// TIA Portal project "FB CONTADOR" (V11)

(* hardware
DEVICE "S7300/ET200 station_1"  SIMATIC 300-Station
   slot 0: "Perfil soporte_0"  Rail  6ES7 390-1***0-0AA0
   slot 1: "PS 307 2A_1"  PS 307 2A  6ES7 307-1BA00-0AA0
   slot 2: "PLC_1"  CPU 313C-2 DP  6ES7 313-6CF03-0AB0  V2.6
      slot 0: "Interfaz MPI_1"  MPI
      slot 1: "Interfaz DP_1"  DP
      slot 2: "DI16/DO16_1"  DI16/DO16
      slot 4: "Contaje_1"  Counter
   slot 4: "AI4/AO2 x 8bits_1"  AI4/AO2x8/8Bit  6ES7 334-0CE01-0AA0
   slot 5: "CP 343-1 Lean_1"  CP 343-1 LEAN  6GK7 343-1CX10-0XE0  V2.4
   slot 6: "CP 340 RS232C_1"  CP 340 RS232C  6ES7 340-1AH02-0AE0  V1.0
   slot 7: "CP 340 RS422/485_2"  CP 340 RS422/485  6ES7 340-1CH02-0AE0  V1.0
*)

// ===== PLC "PLC_1"  CPU 313C-2 DP =====

VAR_GLOBAL   // PLC tag table "Tabla de variables estándar"
   "MARCHA" AT %E0.0 : Bool;
   "PARO" AT %E0.1 : Bool;
   "OUT" AT %A0.0 : Bool;
   "Tag_1" AT %E0.2 : Bool;
   "Tag_2" AT %T0 : Timer;
   "Tag_3" AT %T1 : Timer;
   "Tag_4" AT %I0.3 : Bool;
   "Tag_5" AT %I0.4 : Bool;
   "Tag_6" AT %Q0.1 : Bool;
END_VAR

DATA_BLOCK "CONTADOR_DB"   // DB1
{ S7_Optimized_Access := 'FALSE' }
VERSION : 0.1
// stored: InstanceOfName CONTADOR
"CONTADOR"
BEGIN
END_DATA_BLOCK

DATA_BLOCK "INTERMITENCIA_DB"   // DB2
{ S7_Optimized_Access := 'FALSE' }
VERSION : 0.1
// stored: InstanceOfName INTERMITENCIA
"INTERMITENCIA"
BEGIN
END_DATA_BLOCK

FUNCTION_BLOCK "CONTADOR"   // FB1, LAD
{ S7_Optimized_Access := 'FALSE' }
VERSION : 0.1
   VAR_INPUT
      UP : Bool;
      DOWN : Bool;
      RESET : Bool;
      PV : Real;
      DIGITO : Real;
   END_VAR
   VAR_OUTPUT
      OUT : Bool;
   END_VAR
   VAR
      B0 : Bool;
      B1 : Bool;
      B2 : Bool;
      CONTADOR : Real;
      CONTAJE : Real;
   END_VAR
   VAR_TEMP   // added for the SCL form of the ladder/FBD networks
      _w1 : Bool;
      _w2 : Bool;
   END_VAR
BEGIN

REGION Network 1
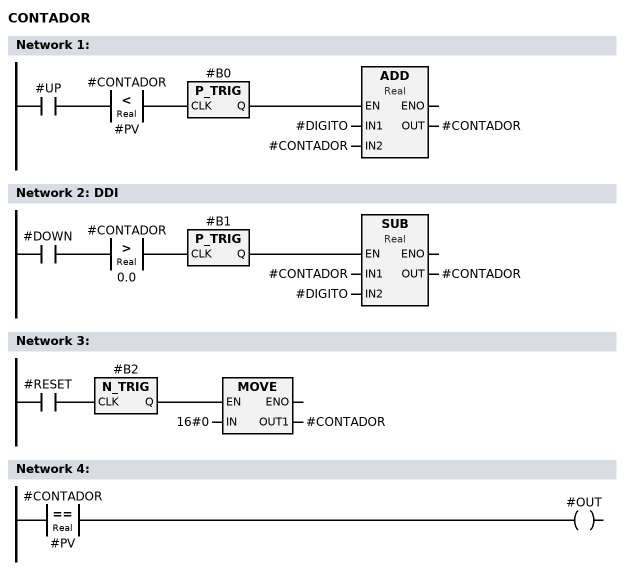
   RUNG wire#powerrail
      Contact( #UP )
      { S7_Templates := "SrcType := Real" } LT_Contact(in1 := #CONTADOR, in2 := #PV)
      P_Trig( #B0 )
      { S7_Templates := "SrcType := Real"; S7_GenerateENO := "TRUE" } Add(in1 := #DIGITO, in2 := #CONTADOR, out => #CONTADOR)
   END_RUNG
   // the same network as SCL:
   #_w1 := #UP AND (#CONTADOR < #PV);
   #_w2 := #_w1 AND NOT #B0;   // rising edge
   #B0 := #_w1;
   IF #_w2 THEN #CONTADOR := #DIGITO + #CONTADOR; END_IF;
END_REGION

REGION Network 2: DDI
   RUNG wire#powerrail
      Contact( #DOWN )
      { S7_Templates := "SrcType := Real" } GT_Contact(in1 := #CONTADOR, in2 := 0.0)
      P_Trig( #B1 )
      { S7_Templates := "SrcType := Real"; S7_GenerateENO := "TRUE" } Sub(in1 := #CONTADOR, in2 := #DIGITO, out => #CONTADOR)
   END_RUNG
   // the same network as SCL:
   #_w1 := #DOWN AND (#CONTADOR > 0.0);
   #_w2 := #_w1 AND NOT #B1;   // rising edge
   #B1 := #_w1;
   IF #_w2 THEN #CONTADOR := #CONTADOR - #DIGITO; END_IF;
END_REGION

REGION Network 3
   RUNG wire#powerrail
      Contact( #RESET )
      N_Trig( #B2 )
      { S7_GenerateENO := "TRUE" } Move(in := 16#0, out1 => #CONTADOR)
   END_RUNG
   // the same network as SCL:
   #_w1 := NOT #RESET AND #B2;   // falling edge
   #B2 := #RESET;
   IF #_w1 THEN #CONTADOR := 16#0; END_IF;
END_REGION

REGION Network 4
   RUNG wire#powerrail
      { S7_Templates := "SrcType := Real" } EQ_Contact(in1 := #CONTADOR, in2 := #PV)
      Coil( #OUT )
   END_RUNG
   // the same network as SCL:
   #OUT := #CONTADOR = #PV;
END_REGION
END_FUNCTION_BLOCK

FUNCTION_BLOCK "INTERMITENCIA"   // FB2, LAD
{ S7_Optimized_Access := 'FALSE' }
VERSION : 0.1
   VAR_INPUT
      "TIM 1" : S5Time;
      "TIM 2" : S5Time;
      TON : Timer;
      TOFF : Timer;
      MARCHA : Bool;
      PARO : Bool;
   END_VAR
   VAR_OUTPUT
      OUT : Bool;
   END_VAR
   VAR
      B0 : Bool;
      B1 : Bool;
      B2 : Bool;
      B3 : Bool;
   END_VAR
BEGIN

REGION Network 1
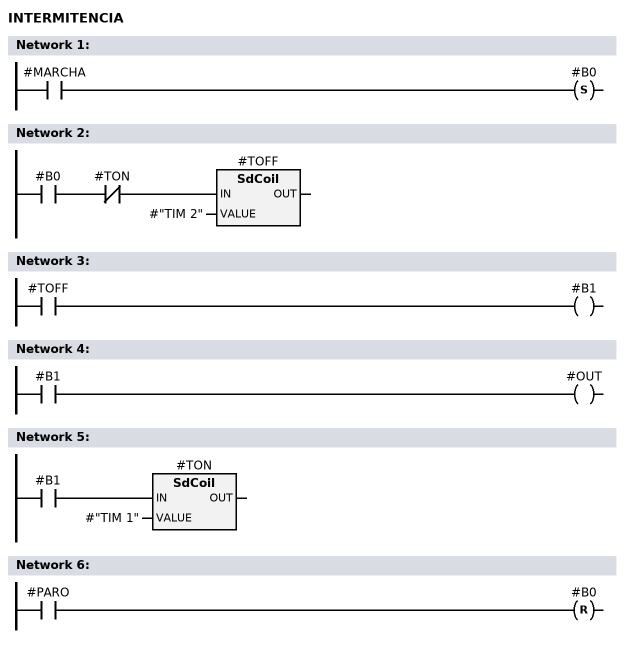
   RUNG wire#powerrail
      Contact( #MARCHA )
      S_Coil( #B0 )
   END_RUNG
   // the same network as SCL:
   IF #MARCHA THEN #B0 := TRUE; END_IF;
END_REGION

REGION Network 2
   // no SCL statement known for SdCoil: written as a call
   SdCoil(in := #B0 AND NOT #TON, value := #"TIM 2", operand := #TOFF);
END_REGION

REGION Network 3
   RUNG wire#powerrail
      Contact( #TOFF )
      Coil( #B1 )
   END_RUNG
   // the same network as SCL:
   #B1 := #TOFF;
END_REGION

REGION Network 4
   RUNG wire#powerrail
      Contact( #B1 )
      Coil( #OUT )
   END_RUNG
   // the same network as SCL:
   #OUT := #B1;
END_REGION

REGION Network 5
   // no SCL statement known for SdCoil: written as a call
   SdCoil(in := #B1, value := #"TIM 1", operand := #TON);
END_REGION

REGION Network 6
   RUNG wire#powerrail
      Contact( #PARO )
      R_Coil( #B0 )
   END_RUNG
   // the same network as SCL:
   IF #PARO THEN #B0 := FALSE; END_IF;
END_REGION
END_FUNCTION_BLOCK

ORGANIZATION_BLOCK "Main"   // OB1, LAD
TITLE = "Main Program Sweep (Cycle)"
{ S7_Optimized_Access := 'FALSE' }
VERSION : 0.1
   VAR_TEMP
      OB1_EV_CLASS : Byte;   // Bits 0-3 = 1 (Coming event), Bits 4-7 = 1 (Event class 1)
      OB1_SCAN_1 : Byte;   // 1 (Cold restart scan 1 of OB 1), 3 (Scan 2-n of OB 1)
      OB1_PRIORITY : Byte;   // Priority of OB Execution
      OB1_OB_NUMBR : Byte;   // 1 (Organization block 1, OB1)
      OB1_RESERVED_1 : Byte;   // Reserved for system
      OB1_RESERVED_2 : Byte;   // Reserved for system
      OB1_PREV_CYCLE : Int;   // Cycle time of previous OB1 scan (milliseconds)
      OB1_MIN_CYCLE : Int;   // Minimum cycle time of OB1 (milliseconds)
      OB1_MAX_CYCLE : Int;   // Maximum cycle time of OB1 (milliseconds)
      OB1_DATE_TIME : Date_And_Time;   // Date and time OB1 started
   END_VAR
BEGIN

REGION Network 1
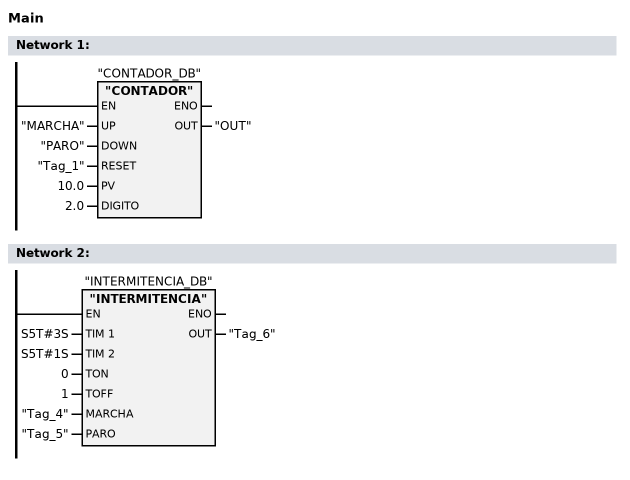
   RUNG wire#powerrail
      "CONTADOR_DB"(UP := "MARCHA", DOWN := "PARO", RESET := "Tag_1", PV := 10.0, DIGITO := 2.0, OUT => "OUT")
   END_RUNG
   // the same network as SCL:
   "CONTADOR_DB"(UP := "MARCHA", DOWN := "PARO", RESET := "Tag_1", PV := 10.0, DIGITO := 2.0, OUT => "OUT");   // "CONTADOR"
END_REGION

REGION Network 2
   RUNG wire#powerrail
      "INTERMITENCIA_DB"("TIM 1" := S5T#3S, "TIM 2" := S5T#1S, TON := 0, TOFF := 1, MARCHA := "Tag_4", PARO := "Tag_5", OUT => "Tag_6")
   END_RUNG
   // the same network as SCL:
   "INTERMITENCIA_DB"("TIM 1" := S5T#3S,   // "INTERMITENCIA"
                      "TIM 2" := S5T#1S,
                      TON := 0,
                      TOFF := 1,
                      MARCHA := "Tag_4",
                      PARO := "Tag_5",
                      OUT => "Tag_6");
END_REGION
END_ORGANIZATION_BLOCK